{attribute addProperty BoxType "EPP6228-0022-0016"}
{attribute addProperty Id "Digital_InputsDigital_Inputs_D24B2EF7648"}
{attribute addProperty CRC "2810777795"}
{attribute addProperty SizeInBites "64"}
{attribute addProperty SizeInBytes "8"}
TYPE Module_11_Digital_Inputs_A78910C3 :
STRUCT
	{attribute addProperty Name "Digital_Inputs"}
	Digital_Inputs  : Digital_Inputs_D24B2EF7;
END_STRUCT
END_TYPE

(* stored: Version 1.2.0.0, ProductVersion 3.1.4024.9
   DUT Module_11_Digital_Inputs_A78910C3: Id {6a54ed80-2719-4e35-beea-906d97559b00} *)
